(* IEC 61131-3 sources: ICSML/Codesys_V3/Function Blocks/LReLU_L.pou, 1 file *)

(* ---- LReLU_L.pou ---- *)
(*#-#-#-#-#-#-#-#-#-#---Declaration---#-#-#-#-#-#-#-#-#-#-#-#-#*)

(*
	Leaky Rectified Linear Unit (LReLU) Activation Layer
*)
FUNCTION_BLOCK PUBLIC LReLU_L IMPLEMENTS Activation
VAR
	// Input and Output dataMem variables
	input_i: dataMem;
	output_i: dataMem;
END_VAR
(*#-#-#-#-#-#-#-#-#-#---Implementation---#-#-#-#-#-#-#-#-#-#-#-#-#*)
